// Mitsubishi GX Works2 project: 14   PLC: FX3G

// task Task_01 (event TRUE, interval 0, priority 31): POU_01

PROGRAM POU_01
VAR
  wstep : INT;
  ton1 : TON;
END_VAR
IF M8002 THEN
	wstep := 0;
END_IF;

CASE wstep OF
	0:
		IF M0 THEN
			wstep := 20;
		END_IF;
	
	20:
		IF M1 THEN
			wstep := 21;
		END_IF;
	
	21:
		Y0 := M8013;
	
		ton1(IN := NOT ton1.Q, PT := T#3s);
		IF ton1.Q THEN
			Y0 := FALSE;
			wstep := 22;
		END_IF;

	22:
		Y1 := TRUE;
		ton1(IN := NOT ton1.Q, PT := T#2s);
		IF ton1.Q THEN
			Y1 := FALSE;
			wstep := 23;
		END_IF;
		
	23:
		Y2 := TRUE;
		IF M2 THEN
			wstep := 24;
		END_IF;
	
	24:
		ton1(IN := NOT ton1.Q, PT := T#5s);
		IF ton1.Q THEN 
			Y2 := FALSE;
			wstep := 20;
		END_IF;
END_CASE;
END_PROGRAM
